PROGRAM PRG_CASE_DuplicateUpdateToDBManual
VAR
	fbCaseDuplicateUpdateToDB		: FB_CASE_DuplicateUpdateToDB;	
END_VAR

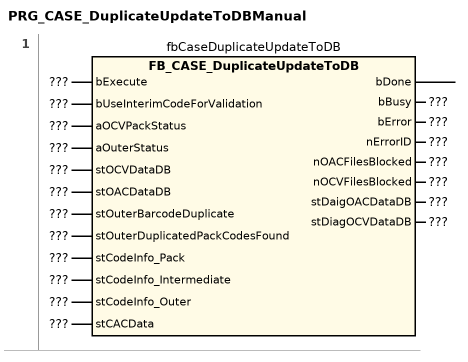
// NETWORK 1
fbCaseDuplicateUpdateToDB(); // FB_CASE_DuplicateUpdateToDB

END_PROGRAM

(* stored: Version 1.1.0.1
   POU PRG_CASE_DuplicateUpdateToDBManual: Id {c89bcf19-9b10-4341-a6c1-b31e3b65bb53}, SpecialFunc None *)
